// TIA Portal V20 export
FUNCTION "Lights" : Void   // FC6, LAD
{ S7_Optimized_Access := 'TRUE' }
// stored: SetENOAutomatically false
   VAR_TEMP
      Column_13_14_CS : Bool;
      Column_14_08_CS : Bool;
      i : SInt;
      Hmi_Button_Drive : Bool;
   END_VAR
BEGIN

REGION Network 1: Safety
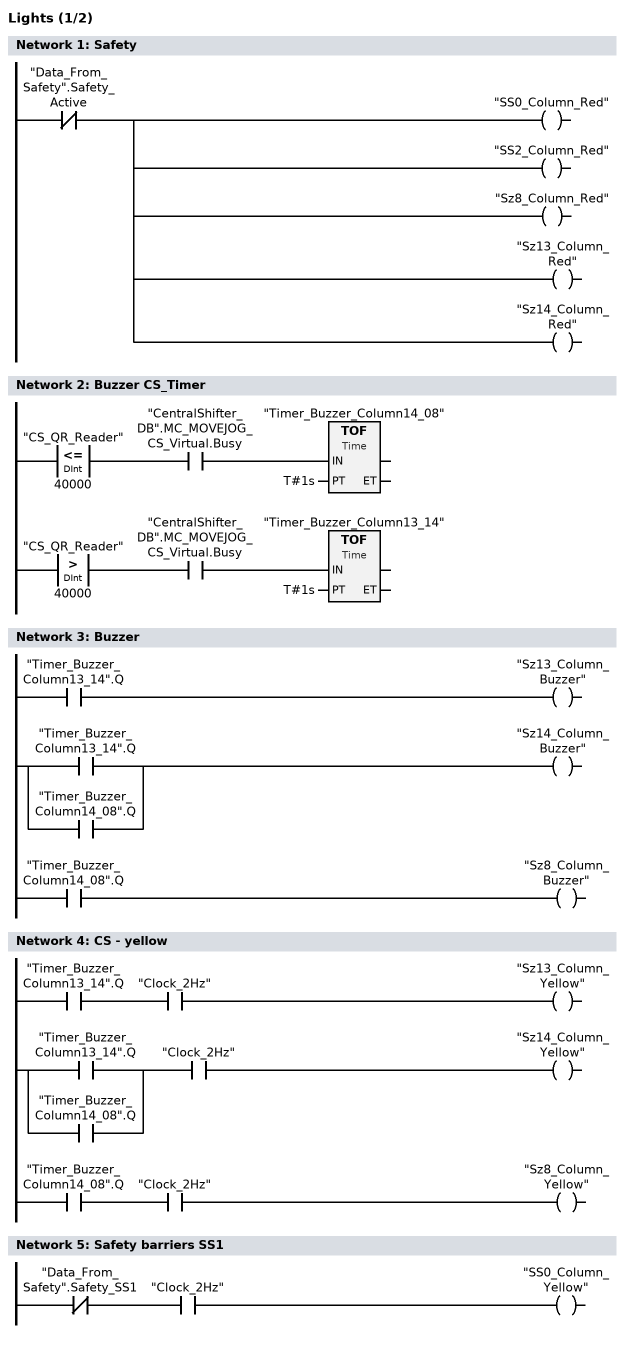
   RUNG wire#powerrail
      I_Contact( "Data_From_Safety".Safety_Active )
      wire#w1
      Coil( "SS0_Column_Red" )
   END_RUNG
   RUNG wire#w1
      Coil( "SS2_Column_Red" )
   END_RUNG
   RUNG wire#w1
      Coil( "Sz8_Column_Red" )
   END_RUNG
   RUNG wire#w1
      Coil( "Sz13_Column_Red" )
   END_RUNG
   RUNG wire#w1
      Coil( "Sz14_Column_Red" )
   END_RUNG
   // the same network as SCL:
   "SS0_Column_Red" := NOT "Data_From_Safety".Safety_Active;
   "SS2_Column_Red" := NOT "Data_From_Safety".Safety_Active;
   "Sz8_Column_Red" := NOT "Data_From_Safety".Safety_Active;
   "Sz13_Column_Red" := NOT "Data_From_Safety".Safety_Active;
   "Sz14_Column_Red" := NOT "Data_From_Safety".Safety_Active;
END_REGION

REGION Network 2: Buzzer CS_Timer
   RUNG wire#powerrail
      { S7_Templates := "SrcType := DInt" } LE_Contact(in1 := "CS_QR_Reader", in2 := 40000)
      Contact( "CentralShifter_DB".MC_MOVEJOG_CS_Virtual.Busy )
      { S7_Templates := "time_type := Time" } "Timer_Buzzer_Column14_08".TOF(pt := T#1s, et =>)
   END_RUNG
   RUNG wire#powerrail
      { S7_Templates := "SrcType := DInt" } GT_Contact(in1 := "CS_QR_Reader", in2 := 40000)
      Contact( "CentralShifter_DB".MC_MOVEJOG_CS_Virtual.Busy )
      { S7_Templates := "time_type := Time" } "Timer_Buzzer_Column13_14".TOF(pt := T#1s, et =>)
   END_RUNG
   // the same network as SCL:
   "Timer_Buzzer_Column14_08".TOF(IN := ("CS_QR_Reader" <= 40000) AND "CentralShifter_DB".MC_MOVEJOG_CS_Virtual.Busy,
                           PT := T#1s);
   "Timer_Buzzer_Column13_14".TOF(IN := ("CS_QR_Reader" > 40000) AND "CentralShifter_DB".MC_MOVEJOG_CS_Virtual.Busy,
                           PT := T#1s);
END_REGION

REGION Network 3: Buzzer
   RUNG wire#powerrail
      Contact( "Timer_Buzzer_Column13_14".Q )
      Coil( "Sz13_Column_Buzzer" )
   END_RUNG
   RUNG wire#powerrail
      Contact( "Timer_Buzzer_Column13_14".Q )
      wire#w1
      Coil( "Sz14_Column_Buzzer" )
   END_RUNG
   RUNG wire#powerrail
      Contact( "Timer_Buzzer_Column14_08".Q )
   END_RUNG wire#w1
   RUNG wire#powerrail
      Contact( "Timer_Buzzer_Column14_08".Q )
      Coil( "Sz8_Column_Buzzer" )
   END_RUNG
   // the same network as SCL:
   "Sz13_Column_Buzzer" := "Timer_Buzzer_Column13_14".Q;
   "Sz14_Column_Buzzer" := "Timer_Buzzer_Column13_14".Q OR "Timer_Buzzer_Column14_08".Q;
   "Sz8_Column_Buzzer" := "Timer_Buzzer_Column14_08".Q;
END_REGION

REGION Network 4: CS - yellow
   RUNG wire#powerrail
      Contact( "Timer_Buzzer_Column13_14".Q )
      Contact( "Clock_2Hz" )
      Coil( "Sz13_Column_Yellow" )
   END_RUNG
   RUNG wire#powerrail
      Contact( "Timer_Buzzer_Column13_14".Q )
      wire#w1
      Contact( "Clock_2Hz" )
      Coil( "Sz14_Column_Yellow" )
   END_RUNG
   RUNG wire#powerrail
      Contact( "Timer_Buzzer_Column14_08".Q )
   END_RUNG wire#w1
   RUNG wire#powerrail
      Contact( "Timer_Buzzer_Column14_08".Q )
      Contact( "Clock_2Hz" )
      Coil( "Sz8_Column_Yellow" )
   END_RUNG
   // the same network as SCL:
   "Sz13_Column_Yellow" := "Timer_Buzzer_Column13_14".Q AND "Clock_2Hz";
   "Sz14_Column_Yellow" := ("Timer_Buzzer_Column13_14".Q OR "Timer_Buzzer_Column14_08".Q) AND "Clock_2Hz";
   "Sz8_Column_Yellow" := "Timer_Buzzer_Column14_08".Q AND "Clock_2Hz";
END_REGION

REGION Network 5: Safety barriers SS1
   RUNG wire#powerrail
      I_Contact( "Data_From_Safety".Safety_SS1 )
      Contact( "Clock_2Hz" )
      Coil( "SS0_Column_Yellow" )
   END_RUNG
   // the same network as SCL:
   "SS0_Column_Yellow" := NOT "Data_From_Safety".Safety_SS1 AND "Clock_2Hz";
END_REGION

REGION Network 6: Safety barrier SS2
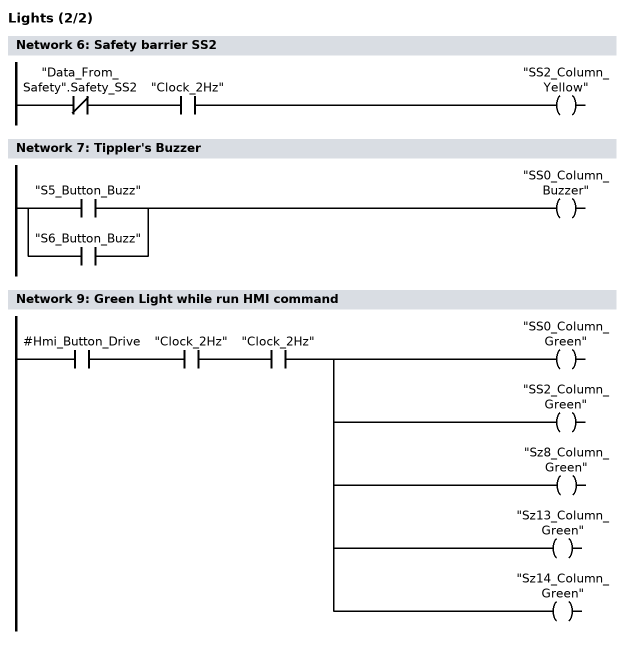
   RUNG wire#powerrail
      I_Contact( "Data_From_Safety".Safety_SS2 )
      Contact( "Clock_2Hz" )
      Coil( "SS2_Column_Yellow" )
   END_RUNG
   // the same network as SCL:
   "SS2_Column_Yellow" := NOT "Data_From_Safety".Safety_SS2 AND "Clock_2Hz";
END_REGION

REGION Network 7: Tippler's Buzzer
   RUNG wire#powerrail
      Contact( "S5_Button_Buzz" )
      wire#w1
      Coil( "SS0_Column_Buzzer" )
   END_RUNG
   RUNG wire#powerrail
      Contact( "S6_Button_Buzz" )
   END_RUNG wire#w1
   // the same network as SCL:
   "SS0_Column_Buzzer" := "S5_Button_Buzz" OR "S6_Button_Buzz";
END_REGION

REGION Network 8 (SCL): Any run button from HMI
       FOR #i := 1 TO 12 DO
           #Hmi_Button_Drive :=
           "HMI_Pallets".Run_Command_left_ROW1[#i] OR
           "HMI_Pallets".Run_Command_left_ROW2[#i] OR
           "HMI_Pallets".Run_Command_left_ROW4[#i] OR
           "HMI_Pallets".Run_Command_right_ROW1[#i] OR
           "HMI_Pallets".Run_Command_right_ROW2[#i] OR
           "HMI_Pallets".Run_Command_right_ROW4[#i];
       END_FOR;
END_REGION

REGION Network 9: Green Light while run HMI command
   RUNG wire#powerrail
      Contact( #Hmi_Button_Drive )
      Contact( "Clock_2Hz" )
      Contact( "Clock_2Hz" )
      wire#w1
      Coil( "SS0_Column_Green" )
   END_RUNG
   RUNG wire#w1
      Coil( "SS2_Column_Green" )
   END_RUNG
   RUNG wire#w1
      Coil( "Sz8_Column_Green" )
   END_RUNG
   RUNG wire#w1
      Coil( "Sz13_Column_Green" )
   END_RUNG
   RUNG wire#w1
      Coil( "Sz14_Column_Green" )
   END_RUNG
   // the same network as SCL:
   "SS0_Column_Green" := #Hmi_Button_Drive AND "Clock_2Hz" AND "Clock_2Hz";
   "SS2_Column_Green" := "SS0_Column_Green";
   "Sz8_Column_Green" := "SS0_Column_Green";
   "Sz13_Column_Green" := "SS0_Column_Green";
   "Sz14_Column_Green" := "SS0_Column_Green";
END_REGION
END_FUNCTION
